(* PLC project CodesysTest_empty.project, CODESYS CODESYS V3.5 SP17 Patch 3 *)
(* stored: creationDateTime 2022-04-22T20:09:13.9279369, modificationDateTime 2022-04-22T11:58:57.9681441 *)

PROGRAM flow1

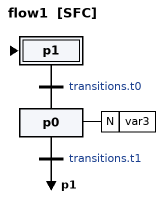
INITIAL_STEP p1:
END_STEP
TRANSITION FROM p1 TO p0
  := transitions.t0;
END_TRANSITION
STEP p0:
  var3(N);
END_STEP
TRANSITION FROM p0 TO p1
  := transitions.t1;
END_TRANSITION
END_PROGRAM
